// TIA Portal V20 export
FUNCTION_BLOCK "FB_AnalogInputs"   // FB220, SCL
{ S7_Optimized_Access := 'FALSE' }
// stored: AutoNumber false, SetENOAutomatically false
   VAR
      sLaserPowerMeter : "FB_AnalogInput";
      sAxisB_ClampingPart : "FB_AnalogInput";
      sLaserAirPressureProcess : "FB_AnalogInput";
      sInletAirPressure : "FB_AnalogInput";
      sAmbiantTemperature : "FB_AnalogInput";
      sMachineTemperature : "FB_AnalogInput";
      sCold_WaterTemperatureInput : "FB_AnalogInput";
      sCold_WaterTemperatureOutput : "FB_AnalogInput";
      sX_AxisTemperaturePT1000 : "FB_AnalogInput";
      sY_AxisTemperaturePT1000 : "FB_AnalogInput";
      sX_AxisTemperaturePTC : "FB_AnalogInput";
      sY_AxisTemperaturePTC : "FB_AnalogInput";
      sNozzleOverpressure : "FB_AnalogInput";
      sOpticalPathOverpressure : "FB_AnalogInput";
      sLaserHeadOverpressure : "FB_AnalogInput";
      sZLAxisOverpressure : "FB_AnalogInput";
      sXYAxisOverpressure : "FB_AnalogInput";
      sLeftAspiration : "FB_AnalogInput";
      sRightAspiration : "FB_AnalogInput";
      sFreeIW458 : "FB_AnalogInput";
      sClimTemperature : "FB_AnalogInput";
      sFreeIW482 : "FB_AnalogInput";
      sFreeIW484 : "FB_AnalogInput";
      sFreeIW486 : "FB_AnalogInput";
      sSensorControllerStation1 : "FB_AnalogInput";
      sCabinetTemperature : "FB_AnalogInput";
      sFreeIW464 : "FB_AnalogInput";
      sFreeIW466 : "FB_AnalogInput";
   END_VAR
   VAR_TEMP
      tAlarm_OutOfRange : Bool;
      tDummyLimit : Real;
   END_VAR
BEGIN
   REGION Description header 
       //==================================================================================
       // POSALUX Swiss SA / (C) Copyright 2025
       //----------------------------------------------------------------------------------
       // Title: Analog Inputs Configuration 
       // Comment/Function: Configuration of analog inputs
       // Author: Fabien WALDT
       // Engineering: TIA Portal v17
       //----------------------------------------------------------------------------------
       // Change log table:
       // Version  | Date     | Expert in charge | Changes applied
       // ---------|----------|------------------|-----------------------------------------
       // 00.00.01 | 20250423 | WFA              | First released version
       // =================================================================================
   END_REGION

   // ET200SP Mapping
   REGION IW412 - IW418 : AI 4xU/I 2-wire ST Slot 9
       #sLaserPowerMeter(iValueHW := "AI_LaserPowerMeter",
                         iID := 701,
                         iHMI_UpdateEnable := TRUE,
                         ioDataHMI := "DB_AnalogInputDataHMI".Laser_Power_Meter,
                         ioAlarmOutOfRange := #tAlarm_OutOfRange,
                         ioDataPLC := "DB_AnalogInputDataPLC".Laser_Power_Meter,
                         ioOPC := "DB_OPC_AnalogInputs".Signals[1]);

       #sAxisB_ClampingPart(iValueHW :="AI_AxisB_ClampingPart",
                            iID:= 810,
                            iHMI_UpdateEnable:= TRUE,
                            ioDataHMI:= "DB_AnalogInputDataHMI".Axis_B_Clamping_Part,
                            ioAlarmOutOfRange := #tAlarm_OutOfRange,
                            ioDataPLC := "DB_AnalogInputDataPLC".Axis_B_Clamping_Part,
                            ioOPC:= "DB_OPC_AnalogInputs".Signals[2]);

       #sLaserAirPressureProcess(iValueHW :="AI_LaserAirPressureProcess",
                                 iID:= 511,
                                 iHMI_UpdateEnable:= TRUE,
                                 ioDataHMI:= "DB_AnalogInputDataHMI".Laser_Air_Pressure_Process,
                                 ioAlarmOutOfRange := #tAlarm_OutOfRange,
                                 ioDataPLC := "DB_AnalogInputDataPLC".Laser_Air_Pressure_Process,
                                 ioOPC:= "DB_OPC_AnalogInputs".Signals[3]);

       #sInletAirPressure(iValueHW :="AI_InletAirPressure",
                          iID:= 501,
                          iHMI_UpdateEnable:= TRUE,
                          ioDataHMI:= "DB_AnalogInputDataHMI".Inlet_Air_Pressure,
                          ioAlarmOutOfRange := "LBP_AlarmMsgs".UserA[01].A70UUxx[03],
                          ioDataPLC := "DB_AnalogInputDataPLC".Inlet_Air_Pressure,
                          ioOPC:= "DB_OPC_AnalogInputs".Signals[4]);
   END_REGION

   REGION IW420 - IW426 : AI4 x RTD/TC HF Slot 10
       #sAmbiantTemperature(iValueHW := "AI_AmbiantTemperature",
                            iID:= 201,
                            iHMI_UpdateEnable:= TRUE,
                            ioDataHMI:= "DB_AnalogInputDataHMI".Ambiant_Temperature,
                            ioAlarmOutOfRange := "LBP_AlarmMsgs".UserA[01].A70UUxx[08],
                            ioDataPLC := "DB_AnalogInputDataPLC".Ambiant_Temperature,
                            ioOPC:= "DB_OPC_AnalogInputs".Signals[5]);

       #sMachineTemperature(iValueHW := "AI_MachineTemperature",
                            iID:= 202,
                            iHMI_UpdateEnable:= TRUE,
                            ioDataHMI:= "DB_AnalogInputDataHMI".Machine_Temperature,
                            ioAlarmOutOfRange := "LBP_AlarmMsgs".UserA[01].A70UUxx[09],
                            ioDataPLC := "DB_AnalogInputDataPLC".Machine_Temperature,
                            ioOPC:= "DB_OPC_AnalogInputs".Signals[6]);

       #sCold_WaterTemperatureInput(iValueHW := "AI_ColdWaterTemperatureInput",
                                    iID:= 301,
                                    iHMI_UpdateEnable:= TRUE,
                                    ioDataHMI:= "DB_AnalogInputDataHMI".Cold_Water_Temperature_Input,
                                    ioAlarmOutOfRange := "LBP_AlarmMsgs".UserA[01].A70UUxx[10],
                                    ioDataPLC := "DB_AnalogInputDataPLC".Cold_Water_Temperature_Input,
                                    ioOPC:= "DB_OPC_AnalogInputs".Signals[7]);

       #sCold_WaterTemperatureOutput(iValueHW := "AI_ColdWaterTemperatureOutput",
                                     iID:= 302,
                                     iHMI_UpdateEnable:= TRUE,
                                     ioDataHMI:= "DB_AnalogInputDataHMI".Cold_Water_Temperature_Output,
                                     ioAlarmOutOfRange := "LBP_AlarmMsgs".UserA[01].A70UUxx[11],
                                     ioDataPLC := "DB_AnalogInputDataPLC".Cold_Water_Temperature_Output,
                                     ioOPC:= "DB_OPC_AnalogInputs".Signals[8]);
   END_REGION

   REGION IW436 - IW442 : AI4 x RTD/TC HF Slot 11
       #sX_AxisTemperaturePT1000(iValueHW := "AI_X_AxisTemperaturePT1000",
                                 iID:= 110,
                                 iHMI_UpdateEnable:= TRUE,
                                 ioDataHMI:= "DB_AnalogInputDataHMI".X_Axis_Temperature_PT1000,
                                 ioAlarmOutOfRange := "LBP_AlarmMsgs".UserA[01].A70UUxx[12],
                                 ioDataPLC := "DB_AnalogInputDataPLC".X_Axis_Temperature_PT1000,
                                 ioOPC:= "DB_OPC_AnalogInputs".Signals[9]);

       #sY_AxisTemperaturePT1000(iValueHW := "AI_Y_AxisTemperaturePT1000",
                                 iID:= 120,
                                 iHMI_UpdateEnable:= TRUE,
                                 ioDataHMI:= "DB_AnalogInputDataHMI".Y_Axis_Temperature_PT1000,
                                 ioAlarmOutOfRange := "LBP_AlarmMsgs".UserA[01].A70UUxx[13],
                                 ioDataPLC := "DB_AnalogInputDataPLC".Y_Axis_Temperature_PT1000,
                                 ioOPC:= "DB_OPC_AnalogInputs".Signals[10]);

       #sX_AxisTemperaturePTC(iValueHW := "AI_X_ AxisTemperaturePTC",
                              iID:= 116,
                              iHMI_UpdateEnable:= TRUE,
                              ioDataHMI:= "DB_AnalogInputDataHMI".X_Axis_Temperature_PTC,
                              ioAlarmOutOfRange := "LBP_AlarmMsgs".UserA[01].A70UUxx[14],
                              ioDataPLC := "DB_AnalogInputDataPLC".X_Axis_Temperature_PTC,
                              ioOPC:= "DB_OPC_AnalogInputs".Signals[11]);

       #sY_AxisTemperaturePTC(iValueHW := "AI_Y_ AxisTemperaturePTC",
                              iID:= 126,
                              iHMI_UpdateEnable:= TRUE,
                              ioDataHMI:= "DB_AnalogInputDataHMI".Y_Axis_Temperature_PTC,
                              ioAlarmOutOfRange := "LBP_AlarmMsgs".UserA[01].A70UUxx[15],
                              ioDataPLC := "DB_AnalogInputDataPLC".Y_Axis_Temperature_PTC,
                              ioOPC:= "DB_OPC_AnalogInputs".Signals[12]);
   END_REGION

   REGION IW444 - IW458 : AI8 x U BA Slot 12
       #sNozzleOverpressure(iValueHW := "AI_NozzleOverpressure",
                            iID:= 512,
                            iHMI_UpdateEnable:= TRUE,
                            ioDataHMI:= "DB_AnalogInputDataHMI".Nozzle_Overpressure,
                            ioAlarmOutOfRange := #tAlarm_OutOfRange,
                            ioDataPLC := "DB_AnalogInputDataPLC".Nozzle_Overpressure,
                            ioOPC:= "DB_OPC_AnalogInputs".Signals[13]);

       #sOpticalPathOverpressure(iValueHW := "AI_OpticalPathOverpressure",
                                 iID:= 513,
                                 iHMI_UpdateEnable:= TRUE,
                                 ioDataHMI:= "DB_AnalogInputDataHMI".Optical_Path_Overpressure,
                                 ioAlarmOutOfRange := "LBP_AlarmMsgs".UserA[01].A70UUxx[05],
                                 ioDataPLC := "DB_AnalogInputDataPLC".Optical_Path_Overpressure,
                                 ioOPC:= "DB_OPC_AnalogInputs".Signals[14]);

       #sLaserHeadOverpressure(iValueHW := "AI_LaserHeadOverpressure",
                               iID:= 514,
                               iHMI_UpdateEnable:= TRUE,
                               ioDataHMI:= "DB_AnalogInputDataHMI".Laser_Head_Overpressure,
                               ioAlarmOutOfRange := "LBP_AlarmMsgs".UserA[01].A70UUxx[06],
                               ioDataPLC := "DB_AnalogInputDataPLC".Laser_Head_Overpressure,
                               ioOPC:= "DB_OPC_AnalogInputs".Signals[15]);

       #sZLAxisOverpressure(iValueHW := "AI_ZL_AxisOverpressure",
                            iID:= 520,
                            iHMI_UpdateEnable:= TRUE,
                            ioDataHMI:= "DB_AnalogInputDataHMI".ZL_Axis_Overpressure,
                            ioAlarmOutOfRange := "LBP_AlarmMsgs".UserA[01].A70UUxx[04],
                            ioDataPLC := "DB_AnalogInputDataPLC".ZL_Axis_Overpressure,
                            ioOPC:= "DB_OPC_AnalogInputs".Signals[16]);

       #sXYAxisOverpressure(iValueHW := "AI_XY_AxisOverpressure",
                            iID:= 530,
                            iHMI_UpdateEnable:= TRUE,
                            ioDataHMI:= "DB_AnalogInputDataHMI".XY_Axis_Overpressure,
                            ioAlarmOutOfRange := "LBP_AlarmMsgs".UserA[01].A70UUxx[07],
                            ioDataPLC := "DB_AnalogInputDataPLC".XY_Axis_Overpressure,
                            ioOPC:= "DB_OPC_AnalogInputs".Signals[17]);

       #sLeftAspiration(iValueHW := "AI_LeftAspiration",
                        iID:= 401,
                        iHMI_UpdateEnable:= TRUE,
                        ioDataHMI:= "DB_AnalogInputDataHMI".Left_Aspiration,
                        ioAlarmOutOfRange := #tAlarm_OutOfRange,
                        ioDataPLC := "DB_AnalogInputDataPLC".Left_Aspiration,
                        ioOPC:= "DB_OPC_AnalogInputs".Signals[18]);

       #sRightAspiration(iValueHW := "AI_RightAspiration",
                         iID:= 402,
                         iHMI_UpdateEnable:= TRUE,
                         ioDataHMI:= "DB_AnalogInputDataHMI".Right_Aspiration,
                         ioAlarmOutOfRange := #tAlarm_OutOfRange,
                         ioDataPLC := "DB_AnalogInputDataPLC".Right_Aspiration,
                         ioOPC:= "DB_OPC_AnalogInputs".Signals[19]);

       #sFreeIW458(iValueHW := "AI_FreeIW458",
                   iID:= 999,
                   iHMI_UpdateEnable:= TRUE,
                   ioDataHMI:= "DB_AnalogInputDataHMI".Free_IW458,
                   ioAlarmOutOfRange := #tAlarm_OutOfRange,
                   ioDataPLC := "DB_AnalogInputDataPLC".Free_IW458,
                   ioOPC:= "DB_OPC_AnalogInputs".Signals[20]);
   END_REGION

   REGION IW480 - IW486 : AI4 x RTD/TC HF Slot 12
       #sClimTemperature(iValueHW := "AI_ClimTemperature",
                         iID:= 204,
                         iHMI_UpdateEnable:= TRUE,
                         ioDataHMI:= "DB_AnalogInputDataHMI".Clim_Temperature,
                         ioAlarmOutOfRange := #tAlarm_OutOfRange,
                         ioDataPLC := "DB_AnalogInputDataPLC".Clim_Temperature,
                         ioOPC:="DB_OPC_AnalogInputs".Signals[21]);

       #sFreeIW482(iValueHW := "AI_FreeIW482",
                   iID:= 999,
                   iHMI_UpdateEnable:=TRUE,
                   ioDataHMI:= "DB_AnalogInputDataHMI".Free_IW482,
                   ioAlarmOutOfRange := #tAlarm_OutOfRange,
                   ioDataPLC := "DB_AnalogInputDataPLC".Free_IW482,
                   ioOPC:= "DB_OPC_AnalogInputs".Signals[22]);

       #sFreeIW484(iValueHW := "AI_FreeIW484",
                   iID:= 999,
                   iHMI_UpdateEnable:= TRUE,
                   ioDataHMI:= "DB_AnalogInputDataHMI".Free_IW484,
                   ioAlarmOutOfRange := #tAlarm_OutOfRange,
                   ioDataPLC := "DB_AnalogInputDataPLC".Free_IW484,
                   ioOPC:= "DB_OPC_AnalogInputs".Signals[23]);

       #sFreeIW486(iValueHW := "AI_FreeIW486",
                   iID:= 999,
                   iHMI_UpdateEnable:= TRUE,
                   ioDataHMI:= "DB_AnalogInputDataHMI".Free_IW486,
                   ioAlarmOutOfRange := #tAlarm_OutOfRange,
                   ioDataPLC := "DB_AnalogInputDataPLC".Free_IW486,
                   ioOPC:= "DB_OPC_AnalogInputs".Signals[24]);
   END_REGION

   REGION IW500 - IW514 : AI 4xU/I 2-wire ST Slot 21
       #sSensorControllerStation1(iValueHW := "AI_SensorControllerStation1",
                                  iID:= 711,
                                  iHMI_UpdateEnable:= TRUE,
                                  ioDataHMI:= "DB_AnalogInputDataHMI".Sensor_Controller_Station1,
                                  ioAlarmOutOfRange := #tAlarm_OutOfRange,
                                  ioDataPLC := "DB_AnalogInputDataPLC".Sensor_Controller_Station1,
                                  ioOPC:= "DB_OPC_AnalogInputs".Signals[25]);

       #sCabinetTemperature(iValueHW := "AI_CabinetTemperature",
                            iID:= 203,
                            iHMI_UpdateEnable:= TRUE,
                            ioDataHMI:= "DB_AnalogInputDataHMI".Cabinet_Temperature,
                            ioAlarmOutOfRange := "LBP_AlarmMsgs".UserA[01].A70UUxx[20],
                            ioDataPLC := "DB_AnalogInputDataPLC".Cabinet_Temperature,
                            ioOPC:= "DB_OPC_AnalogInputs".Signals[26]);

       #sFreeIW464(iValueHW := "AI_FreeIW464",
                   iID:= 999,
                   iHMI_UpdateEnable:= TRUE,
                   ioDataHMI:= "DB_AnalogInputDataHMI".Free_IW464,
                   ioAlarmOutOfRange := #tAlarm_OutOfRange,
                   ioDataPLC := "DB_AnalogInputDataPLC".Free_IW464,
                   ioOPC:= "DB_OPC_AnalogInputs".Signals[27]);

       #sFreeIW466(iValueHW := "AI_FreeIW466",
                   iID:= 999,
                   iHMI_UpdateEnable:= TRUE,
                   ioDataHMI:= "DB_AnalogInputDataHMI".Free_IW466,
                   ioAlarmOutOfRange := #tAlarm_OutOfRange,
                   ioDataPLC := "DB_AnalogInputDataPLC".Free_IW466,
                   ioOPC:= "DB_OPC_AnalogInputs".Signals[28]);
   END_REGION
END_FUNCTION_BLOCK
